// TIA Portal V17 export
// export: Created 2024-09-03T21:55:05.0812472Z, ExportSetting WithDefaults, DisplayName Totally Integrated Automation Portal, DisplayVersion V17 Update 7, DisplayName TIA Portal Openness, DisplayVersion V17 Update 7, DisplayName TIA Portal Version Control Interface, DisplayVersion V17, DisplayName SINAMICS Startdrive Advanced, DisplayVersion V17 SP2, DisplayName SINAMICS Startdrive G110M, G120, G120C, G120D, G120P, G115D, DisplayVersion V17 SP2, DisplayName SINAMICS Startdrive G130, G150, S120, S150, SINAMICS MV, S210, DisplayVersion V17 SP2, DisplayName STEP 7 Professional, DisplayVersion V17 Update 7, DisplayName STEP 7 Safety, DisplayVersion V17 Update 6, DisplayName WinCC Advanced / Unified PC, DisplayVersion V17 Update 7
TYPE "UDT_ConfigEPos"
// stored: IsFailsafeCompliant false
   STRUCT
      Off2 : Bool;
      Off3 : Bool;
      swLimitUsed : Bool;
      hwLimitUsed : Bool;
      reserve1 : Bool;
      reserve2 : Bool;
      reserve3 : Bool;
      reserve4 : Bool;
      reserve5 : Bool;
      reserve6 : Bool;
      reserve7 : Bool;
      reserve8 : Bool;
      reserve9 : Bool;
      reserve10 : Bool;
      reserve11 : Bool;
      reserve12 : Bool;
      reserve13 : Bool;
      reserve14 : Bool;
      reserve15 : Bool;
      reserve16 : Bool;
      reserve17 : Bool;
      reserve18 : Bool;
      reserve19 : Bool;
      reserve20 : Bool;
      reserve21 : Bool;
      reserve22 : Bool;
      reserve23 : Bool;
      reserve24 : Bool;
      reserve25 : Bool;
      reserve26 : Bool;
      reserve27 : Bool;
      reserve28 : Bool;
   END_STRUCT;
END_TYPE
